FUNCTION_BLOCK A_IN (* Service Interface Function Block Type to ESP32 Module *)
  (* Standard: 61499-2; Description: Analog to Digital Converter (ADC) Continuous Mode Driver *)
  (* Version 1.0, 2023-12-13, Filipe Gomes *)
  (* Compiler Cpp Unknown Unknown 1.0 *)
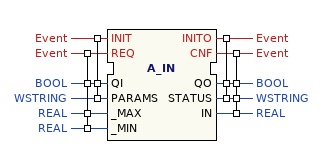
  EVENT_INPUT
    INIT WITH QI, PARAMS; (* Service Initialization *)
    REQ WITH QI, _MAX, _MIN; (* Service Request *)
  END_EVENT
  EVENT_OUTPUT
    INITO WITH QO, STATUS; (* Initialization Confirm *)
    CNF WITH QO, STATUS, IN; (* Confirmation of Requested Service *)
  END_EVENT
  VAR_INPUT
    QI : BOOL := TRUE; (* Event Input Qualifier *)
    PARAMS : WSTRING := ""; (* Pin ID *)
    _MAX : REAL; (* Upper Limit Unit *) {SET_ATTRIBUTE(VarConfig, false)}
    _MIN : REAL; (* Lower Limit Unit *) {SET_ATTRIBUTE(VarConfig, false)}
  END_VAR
  VAR_OUTPUT
    QO : BOOL := FALSE; (* Event Output Qualifier *)
    STATUS : WSTRING := ""; (* Service Status *)
    IN : REAL; (* Input data from resource *)
  END_VAR
  (* Service APPLICATION/RESOURCE: Service Interface Function Block Type to ESP32 Module *)
END_FUNCTION_BLOCK
